{attribute 'c++_compatible'}
///Standard motor
INTERFACE I_StandardMotor EXTENDS I_Object

///Accelaration in FI dependent type
PROPERTY Acc : UINT
GET
END_GET
SET
END_SET
END_PROPERTY

///Move motor CCW
PROPERTY CCW : BOOL
GET
END_GET
SET
END_SET
END_PROPERTY

///Move motor CW
PROPERTY CW : BOOL
GET
END_GET
SET
END_SET
END_PROPERTY

///Deceleration in FI dependent type
PROPERTY Dec : UINT
GET
END_GET
SET
END_SET
END_PROPERTY

///Enable Motor
PROPERTY Enable : BOOL
GET
END_GET
SET
END_SET
END_PROPERTY

///Limit counter-clockwise rotation
PROPERTY LimitCCW : BOOL
GET
END_GET
SET
END_SET
END_PROPERTY

///Limit clockwise rotation
PROPERTY LimitCW : BOOL
GET
END_GET
SET
END_SET
END_PROPERTY

///Pointer to settings, should be set at FB_init but can be modified with set accessor if needed
PROPERTY Settings : POINTER TO ST_StandardMotorSettings
GET
END_GET
SET
END_SET
END_PROPERTY

///Motor speed in 0.1 % 
PROPERTY Speed : UINT
GET
END_GET
SET
END_SET
END_PROPERTY

END_INTERFACE

(* stored: Version 1.1.0.1, ProductVersion 3.1.4019.2
   Itf I_StandardMotor: Id {c80685e9-ce9b-4683-a0af-888a40dbe0c8}
   Folder Settings: Id {f26fb7d2-34ab-42df-b20d-be760832e716}
   Property Acc: Id {aaee8ed9-22dc-4f60-812f-ee60316e8ba1}
   Get Get: Id {63c140a7-fc4d-4c67-a136-8d88382a7505}
   Set Set: Id {8b81c97f-54d6-42e2-b16e-24a8415e6670}
   Property CCW: Id {8d72bd82-8ff5-483b-8cfa-c134cad34dcb}
   Get Get: Id {d2dda53d-70dc-441e-9868-29d19ff844a2}
   Set Set: Id {34a0bbd3-f865-413c-b677-c06918045ea7}
   Property CW: Id {100caab7-60b4-4be3-8c4a-31a315007bc7}
   Get Get: Id {08c3c034-5ea7-46ee-bf50-2f16f0671a1b}
   Set Set: Id {718ba391-32df-4aba-b40f-6840ea9dff1d}
   Property Dec: Id {0ed26595-e6ca-4b99-ba5a-b2b778a818f6}
   Get Get: Id {d751d8a6-d9ad-4f5f-b35a-034d417b96db}
   Set Set: Id {2e1cc78f-756f-48b5-86c3-af68d7688bab}
   Property Enable: Id {64214c29-6dfc-41d1-9de0-b0b89792c952}
   Get Get: Id {487b4847-dbfa-4353-9ee2-9eec4e6981a6}
   Set Set: Id {a067afd7-a885-435e-9f80-37d7837f53d5}
   Property LimitCCW: Id {0fc42405-7106-454f-b1c1-3d4c2fafede4}
   Get Get: Id {f0659a0e-75db-4015-8828-02b23ecc6e82}
   Set Set: Id {92f65689-a42f-4ae5-8aff-20ac800af311}
   Property LimitCW: Id {9a63e3aa-9869-482d-9bf0-912320efc691}
   Get Get: Id {b144c1c7-1985-44e2-bd56-21887061e9e9}
   Set Set: Id {72340fec-a073-4105-baa4-5409dab86888}
   Property Settings: Id {de0bea00-6c90-4466-a84a-0312dd41c133}
   Get Get: Id {ce0ea0d0-e79d-47af-9bee-904f0bba5e68}
   Set Set: Id {1d962c30-10e9-4b07-a20e-38fe81a1342a}
   Property Speed: Id {57f534cb-ca15-42a2-9479-24b55d1d518d}
   Get Get: Id {99d926ae-770a-465b-b58d-3cc84e688080}
   Set Set: Id {3834e235-73ce-4ff9-8667-3346fa9d38c5} *)
